INTERFACE I_MessageData

PROPERTY DirRoot : POINTER to string(255)
SET
END_SET
END_PROPERTY

PROPERTY ErrorIndex : reference to uint
SET
END_SET
END_PROPERTY

PROPERTY FileRoot : pointer to string(255)
SET
END_SET
END_PROPERTY

PROPERTY LocalTime : pointer to DT
SET
END_SET
END_PROPERTY

PROPERTY MessageIndex : reference to uint
SET
END_SET
END_PROPERTY

PROPERTY MsgList : pointer to ARRAY[1..GVL_MSG_XTS.MAX_MESSAGE] OF st_message
SET
END_SET
END_PROPERTY

END_INTERFACE

(* stored: Version 1.1.0.1, ProductVersion 3.1.4026.18
   Itf I_MessageData: Id {47c2a088-e652-443c-88e9-24934af64348}
   Property DirRoot: Id {88024f62-655a-4c0c-a9a5-fb1c5c8b59b9}
   Set Set: Id {3e6e18e5-6e4a-4aad-9567-d38796c5b5d1}
   Property ErrorIndex: Id {c17cda23-74fd-4487-96e1-e87f7fdf95fe}
   Set Set: Id {560e6d4c-2d55-4c6d-9899-7d981d9b4220}
   Property FileRoot: Id {e39d3c25-de33-4b91-b39e-34651c9b84cd}
   Set Set: Id {c35232b0-799b-4c72-8287-bb9c3130e4a8}
   Property LocalTime: Id {ff533578-e4cd-484b-a1ac-737fe16b76d0}
   Set Set: Id {4c20db29-f0d8-4044-bd9e-a0958b793420}
   Property MessageIndex: Id {8a7402cb-53c6-4bca-a9d6-7020c8c9a390}
   Set Set: Id {475664ed-5010-40db-9cc5-0fe45ee1f627}
   Property MsgList: Id {8b304cbf-455b-4b1f-ba47-4582fceb3b66}
   Set Set: Id {6195014a-6766-4f22-a78d-88ba58944820} *)
